{attribute 'linkalways'} 
{attribute 'no_explicit_call' := 'This FB is a CLASS and must be accessed using methods or properties'}
{attribute 'enable_dynamic_creation'}
FUNCTION_BLOCK FINAL EQ_BYTE EXTENDS Node
VAR
	in1 : _BYTE(0);
	in2 : _BYTE(0);
	out : _BOOL(FALSE);
END_VAR

METHOD PUBLIC Clone : I_Node
VAR
	pNode : POINTER TO EQ_BYTE;
END_VAR
pNode := __NEW(EQ_BYTE);
Clone := pNode^;
END_METHOD

METHOD FB_init : BOOL
VAR_INPUT
	bInitRetains : BOOL; // if TRUE, the retain variables are initialized (warm start / cold start)
	bInCopyCode : BOOL;  // if TRUE, the instance afterwards gets moved into the copy code (online change)
END_VAR
AddInput('in1',THIS^.in1);
AddInput('in2',THIS^.in2);
AddOutput('out', THIS^.out);
END_METHOD

METHOD PROTECTED OnExecute
VAR
END_VAR
out.Value := in1.Value = in2.Value;
END_METHOD

END_FUNCTION_BLOCK

(* stored: Version 1.1.0.1, ProductVersion 3.1.4024.15
   POU EQ_BYTE: Id {610be6b2-ce99-4428-bec3-093d41be130a}, SpecialFunc None
   Folder Constructor: Id {d51e76fe-0c29-486b-a106-cf67e3a79e0e}
   Method Clone: Id {72c32ec0-1957-474e-a04c-1984634e56f2}
   Method FB_init: Id {f08f04cb-522d-40f9-899d-1452c2b22a9d}
   Method OnExecute: Id {437ff456-d013-49da-a885-f90fee1bd81a} *)
